# EPICS autosave request: ADApp/Db/NDPluginFile_settings.req
file "NDFile_settings.req",       P=$(P), R=$(R)
file "NDPluginBase_settings.req", P=$(P), R=$(R)
